// TIA Portal V17 export
// export: Created 2022-05-07T16:03:08.7123057Z, ExportSetting WithDefaults, DisplayName Totally Integrated Automation Portal, DisplayVersion V17 Update 3, DisplayName TIA Portal Openness, DisplayVersion V17 Update 3, DisplayName TIA Portal Version Control Interface, DisplayVersion V17, DisplayName TIA Portal Test Suite Advanced, DisplayVersion V17 Update 1, DisplayName SINAMICS Startdrive Advanced, DisplayVersion V17 Update2, DisplayName SINAMICS Startdrive G130, G150, S120, S150, SINAMICS MV, S210, DisplayVersion V17 Update2, DisplayName SINAMICS Startdrive G110M, G120, G120C, G120D, G120P, G115D, DisplayVersion V17 Update2, DisplayName STEP 7 Professional, DisplayVersion V17 Update 3, DisplayName STEP 7 Safety, DisplayVersion V17, DisplayName WinCC UA Professional, DisplayVersion V17 Update 3
FUNCTION_BLOCK "FB_PosizAsseStandard"   // FB2000, LAD
{ S7_Optimized_Access := 'TRUE' }
VERSION : 0.1
// da fare :
// stored: AutoNumber false, IsIECCheckEnabled false, IsRetainMemResEnabled false, MemoryReserve 100, SetENOAutomatically false, UDAEnableTagReadback false
   VAR_INPUT
      Exe_MC_Reset : Bool;   // comando di reset
      En_MC_Power : Bool;   // abilitazione asse
      Exe_MC_Home : Bool;   // comando di homing
      Exe_Jog_Fwd : Bool;   // comando jog +
      Exe_Jog_Rev : Bool;   // comando jog -
      Exe_MC_Velocity : Bool;   // comando velocità
      Exe_MC_Relative : Bool;   // comando posizione relativa
      Exe_MC_Abs : Bool;   // comando posizione assoluta
      Exe_MC_Halt : Bool;   // comando HALT
      Ctl_MC_Stop : Bool;   // comando di controllo STOP
      Sp_lr_MC_HomingOffset : LReal;   // set offset azzeramento (homing)
      Sp_lr_MC_Velocity : LReal;   // set velocità
      Sp_lr_MC_RelativeDistance : LReal;   // set posizione relativa
      Sp_lr_MC_AbsPosition : LReal;   // set posizione assoluta
   END_VAR
   VAR_OUTPUT
      Output_MC_At_Standstill : Bool;   // asse fermo
      Output_MC_AxisEnabled : Bool;
      Output_MC_MoveAbs_Done : Bool;   // move absolute eseguito
      Output_MC_MoveAbs_Busy : Bool;   // move absolute in corso
      Output_MC_Error : Bool;   // asse in errore (or di vari bool)
      Output_MC_AxisHomed : Bool;   // asse homed (referenziato)
      Output_ActVelocity : Real;   // velocity attuale (asse)
      Output_ActPos : Real;   // posizione attuale
   END_VAR
   VAR_IN_OUT
      AxisTO : TO_PositioningAxis;
   END_VAR
   VAR
      AxisReady_PosAxis { S7_SetPoint := 'True'} : Bool;
      MC_Power_Instance_1 { S7_SetPoint := 'True'} : MC_Power;
      MC_Home_Instance_1 { S7_SetPoint := 'True'} : MC_Home;
      MC_MoveJog_Instance_1 { S7_SetPoint := 'True'} : MC_MoveJog;
      MC_MoveVelocity_Instance_1 { S7_SetPoint := 'True'} : MC_MoveVelocity;
      MC_MoveRelative_Instance_1 { S7_SetPoint := 'True'} : MC_MoveRelative;
      MC_MoveAbsolute_Instance_1 { S7_SetPoint := 'True'} : MC_MoveAbsolute;
      MC_Halt_Instance_1 { S7_SetPoint := 'True'} : MC_Halt;
      MC_Reset_Instance_1 { S7_SetPoint := 'True'} : MC_Reset;
   END_VAR
   VAR CONSTANT
      VALID : DInt := 2;
      ADAPTED : DInt := 2;
      NOT_APPLICABLE : DInt := 3;
   END_VAR
BEGIN

REGION Network 1: MC_RESET
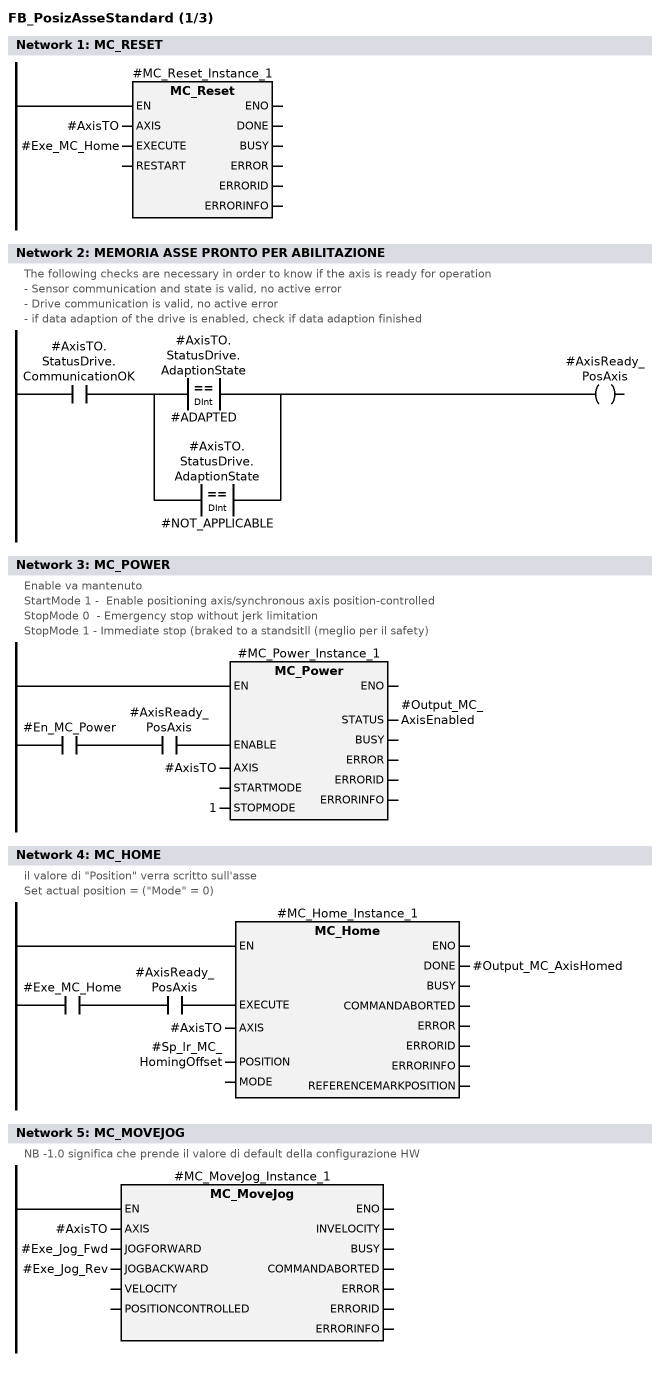
   RUNG wire#powerrail
      #MC_Reset_Instance_1.MC_Reset(Axis := #AxisTO, Execute := #Exe_MC_Home, Restart :=, Done =>, Busy =>, Error =>, ErrorID =>, ErrorInfo =>)
   END_RUNG
   // the same network as SCL:
   #MC_Reset_Instance_1(Axis := #AxisTO, Execute := #Exe_MC_Home);   // MC_Reset
END_REGION

REGION Network 2: MEMORIA ASSE PRONTO PER ABILITAZIONE
   // The following checks are necessary in order to know if the axis is ready for operation
   // - Sensor communication and state is valid, no active error
   // - Drive communication is valid, no active error
   // - if data adaption of the drive is enabled, check if data adaption finished
   RUNG wire#powerrail
      Contact( #AxisTO.StatusDrive.CommunicationOK )
      wire#w1
      { S7_Templates := "SrcType := DInt" } EQ_Contact(in1 := #AxisTO.StatusDrive.AdaptionState, in2 := #ADAPTED)
      wire#w2
      Coil( #AxisReady_PosAxis )
   END_RUNG
   RUNG wire#w1
      { S7_Templates := "SrcType := DInt" } EQ_Contact(in1 := #AxisTO.StatusDrive.AdaptionState, in2 := #NOT_APPLICABLE)
   END_RUNG wire#w2
   // the same network as SCL:
   #AxisReady_PosAxis := #AxisTO.StatusDrive.CommunicationOK AND ((#AxisTO.StatusDrive.AdaptionState = #ADAPTED) OR (#AxisTO.StatusDrive.AdaptionState = #NOT_APPLICABLE));
END_REGION

REGION Network 3: MC_POWER
   // Enable va mantenuto
   // StartMode 1 - ​​ Enable positioning axis/synchronous axis position-controlled
   // StopMode 0  - Emergency stop without jerk limitation
   // StopMode 1 - ​Immediate stop (braked to a standsitll (meglio per il safety)
   RUNG wire#powerrail
      #MC_Power_Instance_1.MC_Power(Enable := wire#w1, Axis := #AxisTO, StartMode :=, StopMode := 1, Status => #Output_MC_AxisEnabled, Busy =>, Error =>, ErrorID =>, ErrorInfo =>)
   END_RUNG
   RUNG wire#powerrail
      Contact( #En_MC_Power )
      Contact( #AxisReady_PosAxis )
   END_RUNG wire#w1
   // the same network as SCL:
   #MC_Power_Instance_1(Enable := #En_MC_Power AND #AxisReady_PosAxis,   // MC_Power
                        Axis := #AxisTO,
                        StopMode := 1,
                        Status => #Output_MC_AxisEnabled);
END_REGION

REGION Network 4: MC_HOME
   // il valore di "Position" verra scritto sull'asse
   // Set actual position = ("Mode" = 0)
   RUNG wire#powerrail
      #MC_Home_Instance_1.MC_Home(Execute := wire#w1, Axis := #AxisTO, Position := #Sp_lr_MC_HomingOffset, Mode :=, Done => #Output_MC_AxisHomed, Busy =>, CommandAborted =>, Error =>, ErrorID =>, ErrorInfo =>, ReferenceMarkPosition =>)
   END_RUNG
   RUNG wire#powerrail
      Contact( #Exe_MC_Home )
      Contact( #AxisReady_PosAxis )
   END_RUNG wire#w1
   // the same network as SCL:
   #MC_Home_Instance_1(Execute := #Exe_MC_Home AND #AxisReady_PosAxis,   // MC_Home
                       Axis := #AxisTO,
                       Position := #Sp_lr_MC_HomingOffset,
                       Done => #Output_MC_AxisHomed);
END_REGION

REGION Network 5: MC_MOVEJOG
   // NB -1.0 significa che prende il valore di default della configurazione HW
   RUNG wire#powerrail
      #MC_MoveJog_Instance_1.MC_MoveJog(Axis := #AxisTO, JogForward := #Exe_Jog_Fwd, JogBackward := #Exe_Jog_Rev, Velocity :=, PositionControlled :=, InVelocity =>, Busy =>, CommandAborted =>, Error =>, ErrorID =>, ErrorInfo =>)
   END_RUNG
   // the same network as SCL:
   #MC_MoveJog_Instance_1(Axis := #AxisTO, JogForward := #Exe_Jog_Fwd, JogBackward := #Exe_Jog_Rev);   // MC_MoveJog
END_REGION

REGION Network 6: MC_MOVEVELOCITY
   // per gerstire l'asse in controllo velocità
   // per fermarlo usare HALT oppure STOP
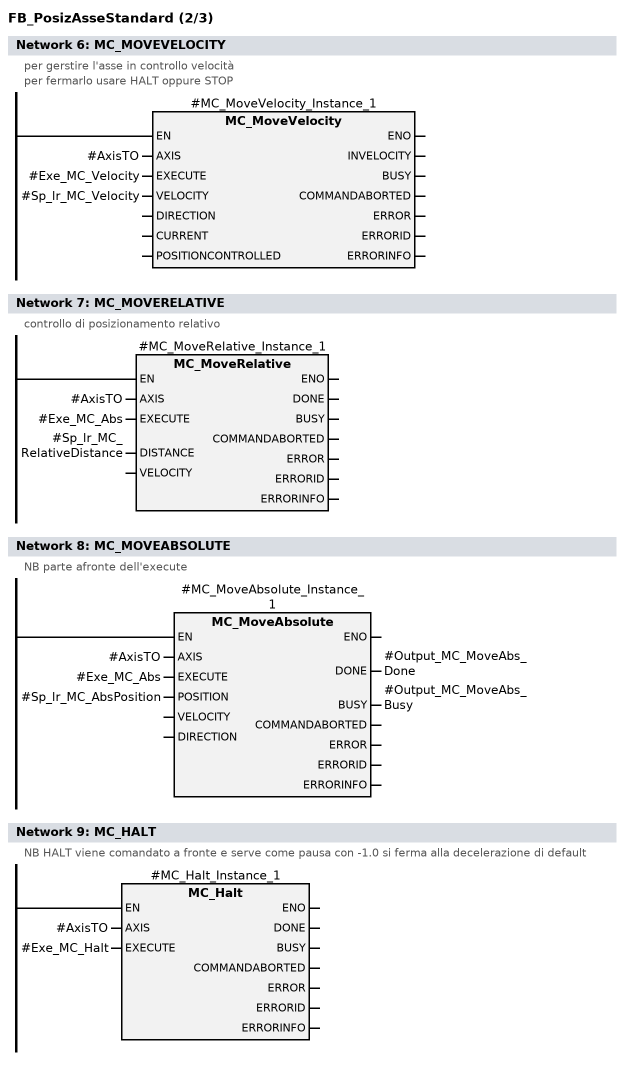
   RUNG wire#powerrail
      #MC_MoveVelocity_Instance_1.MC_MoveVelocity(Axis := #AxisTO, Execute := #Exe_MC_Velocity, Velocity := #Sp_lr_MC_Velocity, Direction :=, Current :=, PositionControlled :=, InVelocity =>, Busy =>, CommandAborted =>, Error =>, ErrorID =>, ErrorInfo =>)
   END_RUNG
   // the same network as SCL:
   #MC_MoveVelocity_Instance_1(Axis := #AxisTO, Execute := #Exe_MC_Velocity, Velocity := #Sp_lr_MC_Velocity);   // MC_MoveVelocity
END_REGION

REGION Network 7: MC_MOVERELATIVE
   // controllo di posizionamento relativo
   RUNG wire#powerrail
      #MC_MoveRelative_Instance_1.MC_MoveRelative(Axis := #AxisTO, Execute := #Exe_MC_Abs, Distance := #Sp_lr_MC_RelativeDistance, Velocity :=, Done =>, Busy =>, CommandAborted =>, Error =>, ErrorID =>, ErrorInfo =>)
   END_RUNG
   // the same network as SCL:
   #MC_MoveRelative_Instance_1(Axis := #AxisTO, Execute := #Exe_MC_Abs, Distance := #Sp_lr_MC_RelativeDistance);   // MC_MoveRelative
END_REGION

REGION Network 8: MC_MOVEABSOLUTE
   // NB parte afronte dell'execute
   RUNG wire#powerrail
      #MC_MoveAbsolute_Instance_1.MC_MoveAbsolute(Axis := #AxisTO, Execute := #Exe_MC_Abs, Position := #Sp_lr_MC_AbsPosition, Velocity :=, Direction :=, Done => #Output_MC_MoveAbs_Done, Busy => #Output_MC_MoveAbs_Busy, CommandAborted =>, Error =>, ErrorID =>, ErrorInfo =>)
   END_RUNG
   // the same network as SCL:
   #MC_MoveAbsolute_Instance_1(Axis := #AxisTO,   // MC_MoveAbsolute
                           Execute := #Exe_MC_Abs,
                           Position := #Sp_lr_MC_AbsPosition,
                           Done => #Output_MC_MoveAbs_Done,
                           Busy => #Output_MC_MoveAbs_Busy);
END_REGION

REGION Network 9: MC_HALT
   // NB HALT viene comandato a fronte e serve come pausa con -1.0 si ferma alla decelerazione di default
   RUNG wire#powerrail
      #MC_Halt_Instance_1.MC_Halt(Axis := #AxisTO, Execute := #Exe_MC_Halt, Done =>, Busy =>, CommandAborted =>, Error =>, ErrorID =>, ErrorInfo =>)
   END_RUNG
   // the same network as SCL:
   #MC_Halt_Instance_1(Axis := #AxisTO, Execute := #Exe_MC_Halt);   // MC_Halt
END_REGION

REGION Network 10: VALORI ATTUALI
   // speed = vel motore 
   // velocity = vel asse
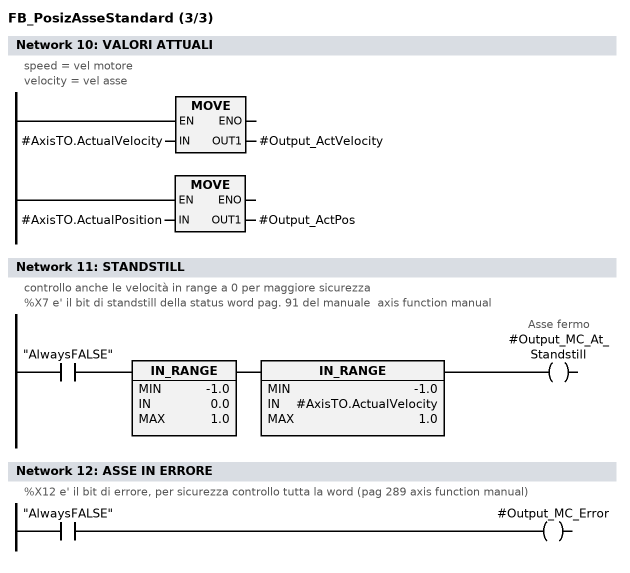
   RUNG wire#powerrail
      Move(in := #AxisTO.ActualVelocity, out1 => #Output_ActVelocity)
   END_RUNG
   RUNG wire#powerrail
      Move(in := #AxisTO.ActualPosition, out1 => #Output_ActPos)
   END_RUNG
   // the same network as SCL:
   #Output_ActVelocity := #AxisTO.ActualVelocity;
   #Output_ActPos := #AxisTO.ActualPosition;
END_REGION

REGION Network 11: STANDSTILL
   // controllo anche le velocità in range a 0 per maggiore sicurezza
   // %X7 e' il bit di standstill della status word pag. 91 del manuale  axis function manual
   RUNG wire#powerrail
      Contact( "AlwaysFALSE" )
      { S7_Templates := "SrcType := LReal" } InRange(min := -1.0, in := 0.0, max := 1.0)
      { S7_Templates := "SrcType := LReal" } InRange(min := -1.0, in := #AxisTO.ActualVelocity, max := 1.0)
      Coil( #Output_MC_At_Standstill )   // Asse fermo
   END_RUNG
   // the same network as SCL:
   #Output_MC_At_Standstill := "AlwaysFALSE" AND (-1.0 <= 0.0) AND (0.0 <= 1.0) AND (-1.0 <= #AxisTO.ActualVelocity) AND (#AxisTO.ActualVelocity <= 1.0);   // Asse fermo
END_REGION

REGION Network 12: ASSE IN ERRORE
   // %X12 e' il bit di errore, per sicurezza controllo tutta la word (pag 289 axis function manual)
   RUNG wire#powerrail
      Contact( "AlwaysFALSE" )
      Coil( #Output_MC_Error )
   END_RUNG
   // the same network as SCL:
   #Output_MC_Error := "AlwaysFALSE";
END_REGION
END_FUNCTION_BLOCK
